(* PLC project Unnamed, Unknown Unnamed 1 *)
(* stored: creationDateTime 2023-03-10T10:37:17, modificationDateTime 2023-03-23T23:20:19 *)

(* SIEMENS AG- Beispielprogramm *)
FUNCTION_BLOCK Shop_Window_Lighting
  VAR_INPUT
    IN1 : BOOL;
    IN2 : BOOL;
    IN3 : BOOL;
    IN4 : BOOL;
    TIME3 : BOOL;
  END_VAR
  VAR_OUTPUT
    OUT1 : BOOL;
    OUT2 : BOOL;
    OUT3 : BOOL;
    OUT4 : BOOL;
  END_VAR
  VAR
    TOF0 : TOF;
    TOF1 : TOF;
    PT1m : TIME;
  END_VAR
  VAR  (* added by the conversion: wires and edge detectors of the diagram *)
    _AND2_OUT : BOOL;
  END_VAR

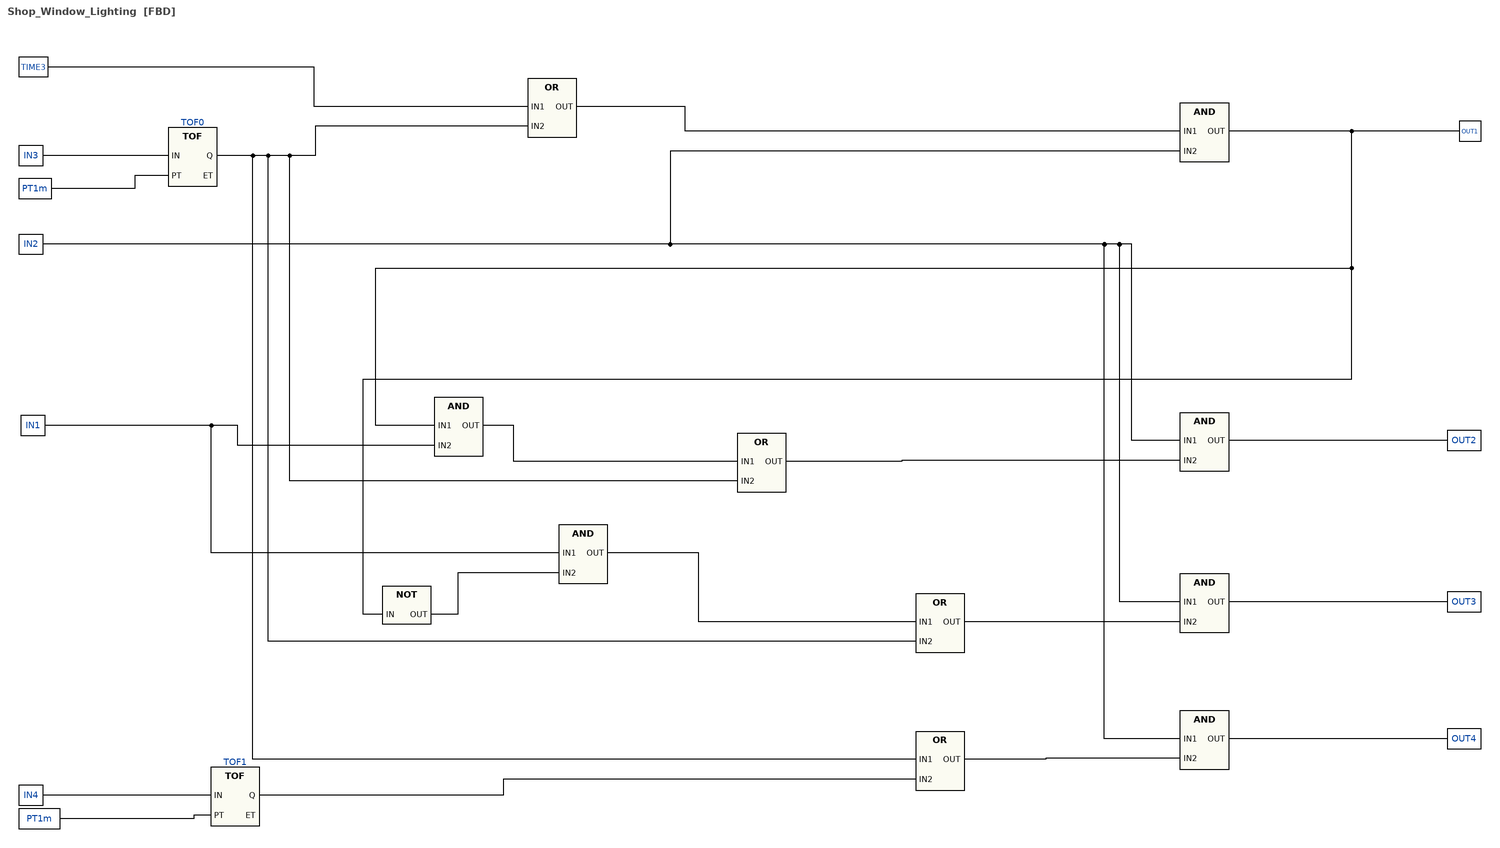
(* FBD diagram, written out as Structured Text *)
TOF0(IN := IN3, PT := PT1m);
_AND2_OUT := (TIME3 OR TOF0.Q) AND IN2;
OUT1 := _AND2_OUT;
OUT2 := IN2 AND (_AND2_OUT AND IN1 OR TOF0.Q);
OUT3 := IN2 AND (IN1 AND NOT _AND2_OUT OR TOF0.Q);
TOF1(IN := IN4, PT := PT1m);
OUT4 := IN2 AND (TOF0.Q OR TOF1.Q);
END_FUNCTION_BLOCK

CONFIGURATION config
  RESOURCE resource1 ON PLC
  END_RESOURCE
END_CONFIGURATION
